PROGRAM MAIN
VAR
END_VAR

END_PROGRAM

(* stored: Version 1.1.0.1
   POU MAIN: Id {72747298-b432-40d1-a6ee-50fb1c1d239f} *)
